FUNCTION Convert_BOOL_TO_ULINT : BOOL
VAR_INPUT
	in : BOOL;
	out : REFERENCE TO ULINT;
END_VAR
VAR
	converted : ULINT;
END_VAR

converted := BOOL_TO_ULINT(in);

IF (ULINT_TO_BOOL(converted) <> in) THEN
	RETURN;
END_IF

out := converted;
Convert_BOOL_TO_ULINT := TRUE;

END_FUNCTION

(* stored: Version 1.1.0.1, ProductVersion 3.1.4024.12
   POU Convert_BOOL_TO_ULINT: Id {839a4765-1b45-4f2e-a7fa-2adfaf8521b1}, SpecialFunc None *)
